ABB RobotStudio station: Estacion_Proyecto.rsstn

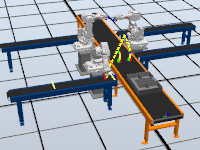
Station Station (saved by RobotStudio 20.4.9280.0)
Controller Controlador_Vajilla
  mechanical unit ROB_1: IRB140_6_81_C_03_1, 6 joints, base frame (0, 570, 550) mm, rotated rx 0 ry 0 rz -90 deg
  mechanical unit ROB_2: IRB140_6_81_C_03_2, 6 joints, base frame (1000, 570, 550) mm, rotated rx 0 ry 0 rz -90 deg
  mechanical unit ROB_3: IRB140_6_81_C_03_3, 6 joints, base frame (850, -570, 550) mm, rotated rx 0 ry 0 rz 90 deg
Layout (positions relative to the parent item):
  - set de 6 puestos-caja [part] at (-1002.05, -1.51, 606.8) mm, rotated rx 0 ry 0 rz 179.54 deg
  - set de 6 puestos-plato_hondo [part] at (-543.94, 2197.29, 0) mm, rotated rx -0.11 ry 0 rz 0 deg
  - set de 6 puestos-plato_pando [part]
  - set de 6 puestos-plato_postre [part]
  - set de 6 puestos-vaso [part] at (1.15, 0.93, 0.79) mm, rotated rx 0 ry 0 rz 0.13 deg
  - IRB140_6_81_C_03_1 [mechanism, from Robots\IRB140_6_81_C_G_03.rslib] at (0, 570, 550) mm, rotated rx 0 ry 0 rz -90 deg; joint values [-1.5708, 0.9264, 0.1141, 0, 0.5303, -1.5708] (rad or m)
  - IRB140_6_81_C_03_2 [mechanism, from Robots\IRB140_6_81_C_G_03.rslib] at (1000, 570, 550) mm, rotated rx 0 ry 0 rz -90 deg; joint values [0, 0, 0, 0.0533, 0.5236, 0] (rad or m)
  - IRB140_6_81_C_03_3 [mechanism, from Robots\IRB140_6_81_C_G_03.rslib] at (850, -570, 550) mm, rotated rx 0 ry 0 rz 90 deg; joint values [0, 0, 0, 0, 0.5236, 0] (rad or m)
  - Sockel_IRB140_500mm_3 [part, from Proyecto\53244bc2-0fdb-48b8-abaf-b031e49cfeeesockel_irb140_500mm.rslib] at (850, -570, 0) mm, rotated rx 0 ry 0 rz 90 deg
  - Sockel_IRB140_500mm_1 [part, from Proyecto\53244bc2-0fdb-48b8-abaf-b031e49cfeeesockel_irb140_500mm.rslib] at (0, 570, 0) mm, rotated rx 0 ry 0 rz -90 deg
  - Sockel_IRB140_500mm_2 [part, from Proyecto\53244bc2-0fdb-48b8-abaf-b031e49cfeeesockel_irb140_500mm.rslib] at (1000, 570, 0) mm, rotated rx 0 ry 0 rz -90 deg
  - Linea_Plato_Pando [part]
  - Linea_Plato_Postre [part]
  - Linea_Plato_Hondo [part]
  - Linea_Vaso [part]
  - Linea_Principal [part]
  - VacuumToolCreator [smart component, from Proyecto\d28571e4-d633-4a15-b430-832653a4066fvacuumtoolcreator.rslib]
      properties: Tool Name=VacuumTool; TCP Name=tVacuum; TCP Position=[0 0 0.049]; TCP Orientation=[0 0 0]; Flange Diameter=0.055; Length=0.1; Width=0.1; Solids only=false; GeneratedTool=VacuumTool
  - VacuumTool [mechanism] at (-550, 570, 725.45) mm, rotated rx -180 ry 0 rz 90 deg
      TCP tVacuum at (0, 0, 49) mm
      links: VacuumTool
  - SmartComponent_1 [smart component]
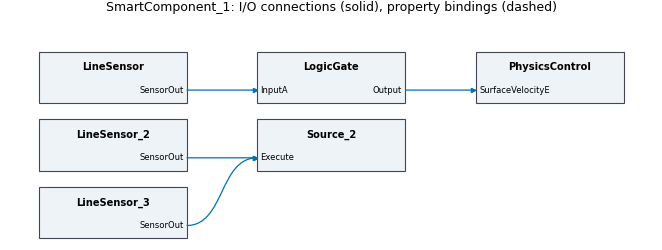
      connections:
        LineSensor.SensorOut -> LogicGate.InputA
        LogicGate.Output -> PhysicsControl.SurfaceVelocityEnabled
        LineSensor_2.SensorOut -> Source_2.Execute
        LineSensor_3.SensorOut -> Source_2.Execute
    - Source_2 [smart component, from Components\Source.rslib] at (-390.95, 79.72, -105.31) mm, rotated rx 0 ry 0 rz -28.76 deg
        properties: Source=set de 6 puestos-plato_hondo; Copy=(none); Parent=(none); Position=[-0.55 2.2 0.6]; Orientation=[0 0 0]; Transient=true; PhysicsBehavior=3
    - LineSensor [smart component, from Components\LineSensor.rslib]
        properties: Start=[-0.4 0.46 0.6405]; End=[-0.7 0.46 0.6405]; Radius=0.004; SensedPart=(none); SensedPoint=[0 0 0]
      - _sensorPart_ [part]
    - PhysicsControl [smart component, from Components\PhysicsControl.rslib]
        properties: Object=Linea_Plato_Hondo; Behavior=1; SurfaceVelocity=0.1
    - LogicGate [smart component, from Components\LogicGate.rslib]
        properties: Operator=NOT; Delay=0
    - LineSensor_3 [smart component, from Components\LineSensor.rslib]
        properties: Start=[-0.4 1.6 0.6405]; End=[-0.7 1.6 0.6405]; Radius=0.004; SensedPart=(none); SensedPoint=[0 0 0]
      - _sensorPart_ [part]
Attachment: VacuumTool is attached to IRB140_6_81_C_03_1 / Link6
Attachment: Sockel_IRB140_500mm_3 is attached to IRB140_6_81_C_03_3 / Base
Attachment: Sockel_IRB140_500mm_1 is attached to IRB140_6_81_C_03_1 / Base
Attachment: Sockel_IRB140_500mm_2 is attached to IRB140_6_81_C_03_2 / Base
Attachment: Source_2 is attached to IRB140_6_81_C_03_1 / Link6
Attachment: PhysicsControl is attached to Sockel_IRB140_500mm_2
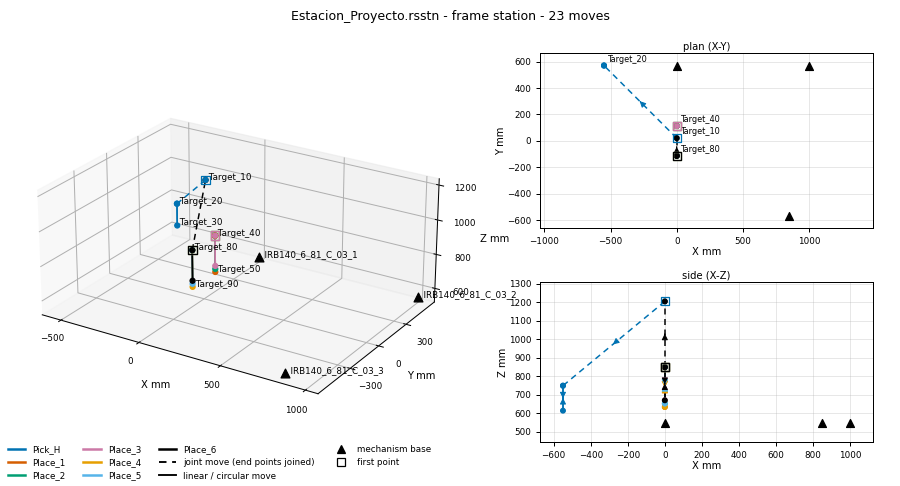
[picture p0: tool path of Estacion_Proyecto.rsstn in frame station, 23 of 23 moves have a stored position in this frame; points joined in program order, loops and branches not executed]
Targets, tools, work objects and paths stored in the station, written as RAPID:
! task T_ROB1
MODULE CalibData
  PERS tooldata tVacuum:=[TRUE,[[0,0,49],[1,0,0,0]],[1,[0,0,32.666666667],[1,0,0,0],0,0,0]];
  TASK PERS wobjdata PlatoH:=[FALSE,TRUE,"",[[-550,400,600],[1,0,0,0]],[[0,0,0],[1,0,0,0]]];
  TASK PERS wobjdata Principal:=[FALSE,TRUE,"",[[-2000,0,600],[1,0,0,0]],[[0,0,0],[1,0,0,0]]];
ENDMODULE

! task T_ROB1
MODULE Module1
  CONST robtarget Target_10:=[[550,-378.726896031,605],[0.353553391,0.612372436,0.612372436,-0.353553391],[0,0,0,0],[9E+09,9E+09,9E+09,9E+09,9E+09,9E+09]];
  CONST robtarget Target_20:=[[-0.000010331,170.000024041,150.000000196],[-0.000000016,0.707106781,0.707106781,-0.000000016],[-2,0,-2,0],[9E+09,9E+09,9E+09,9E+09,9E+09,9E+09]];
  CONST robtarget Target_30:=[[0,170,15],[0,0.707106781,0.707106781,0],[-2,-1,-2,0],[9E+09,9E+09,9E+09,9E+09,9E+09,9E+09]];
  CONST robtarget Target_40:=[[2000,112.500025345,250.0000139],[0,-0.004974188,0.999987629,-0.000000008],[0,-1,-2,0],[9E+09,9E+09,9E+09,9E+09,9E+09,9E+09]];
  CONST robtarget Target_50:=[[2000,112.499986498,34.999992831],[0,-0.004974188,0.999987629,-0.000000038],[0,-1,-2,0],[9E+09,9E+09,9E+09,9E+09,9E+09,9E+09]];
  CONST robtarget Target_60:=[[2000,112.500003859,52.999957808],[0,-0.004974188,0.999987629,0.000000022],[-1,0,-2,0],[9E+09,9E+09,9E+09,9E+09,9E+09,9E+09]];
  CONST robtarget Target_70:=[[2000,112.5,71],[0,-0.004974168,0.999987629,0],[0,-1,-2,0],[9E+09,9E+09,9E+09,9E+09,9E+09,9E+09]];
  CONST robtarget Target_80:=[[2000,-112.5,250],[0,-0.004974168,0.999987629,0],[0,-1,-2,0],[9E+09,9E+09,9E+09,9E+09,9E+09,9E+09]];
  CONST robtarget Target_90:=[[2000,-112.5,35],[0,-0.004974168,0.999987629,0],[0,0,-2,0],[9E+09,9E+09,9E+09,9E+09,9E+09,9E+09]];
  CONST robtarget Target_100:=[[2000,-112.5,53],[0,-0.004974168,0.999987629,0],[0,0,-2,0],[9E+09,9E+09,9E+09,9E+09,9E+09,9E+09]];
  CONST robtarget Target_110:=[[2000,-112.5,71],[0,-0.004974168,0.999987629,0],[0,0,-2,0],[9E+09,9E+09,9E+09,9E+09,9E+09,9E+09]];
  PROC Pick_H()
    MoveJ Target_10,v1000,z10,tVacuum\WObj:=PlatoH;
    MoveJ Target_20,v1000,z10,tVacuum\WObj:=PlatoH;
    MoveL Target_30,v80,z10,tVacuum\WObj:=PlatoH;
    MoveL Target_20,v80,z10,tVacuum\WObj:=PlatoH;
  ENDPROC
  PROC Place_1()
    MoveL Target_40,v200,z10,tVacuum\WObj:=Principal;
    MoveL Target_50,v80,z10,tVacuum\WObj:=Principal;
    MoveL Target_40,v80,z10,tVacuum\WObj:=Principal;
  ENDPROC
  PROC Place_2()
    MoveL Target_40,v200,z10,tVacuum\WObj:=Principal;
    MoveL Target_60,v80,z10,tVacuum\WObj:=Principal;
    MoveL Target_40,v80,z10,tVacuum\WObj:=Principal;
  ENDPROC
  PROC Place_3()
    MoveL Target_40,v200,z10,tVacuum\WObj:=Principal;
    MoveL Target_70,v80,z10,tVacuum\WObj:=Principal;
    MoveL Target_40,v80,z10,tVacuum\WObj:=Principal;
  ENDPROC
  PROC Place_4()
    MoveL Target_80,v200,z10,tVacuum\WObj:=Principal;
    MoveL Target_90,v80,z10,tVacuum\WObj:=Principal;
    MoveL Target_80,v80,z10,tVacuum\WObj:=Principal;
  ENDPROC
  PROC Place_5()
    MoveL Target_80,v200,z10,tVacuum\WObj:=Principal;
    MoveL Target_100,v80,z10,tVacuum\WObj:=Principal;
    MoveL Target_80,v80,z10,tVacuum\WObj:=Principal;
  ENDPROC
  PROC Place_6()
    MoveL Target_80,v200,z10,tVacuum\WObj:=Principal;
    MoveL Target_110,v80,z10,tVacuum\WObj:=Principal;
    MoveL Target_80,v80,z10,tVacuum\WObj:=Principal;
    MoveJ Target_10,v1000,z10,tVacuum\WObj:=PlatoH;
  ENDPROC
  PROC main()
    Pick_H;
    Place_1;
    Pick_H;
    Place_2;
    Pick_H;
    Place_3;
    Pick_H;
    Place_4;
    Pick_H;
    Place_5;
    Pick_H;
    Place_6;
  ENDPROC
ENDMODULE

